PROGRAM ControlePID_Ladder
  VAR
    NIVEL_PV_RAW : UINT := 0;
    AUX_NIVEL_PV : REAL := 0;
    AUX_NIVEL_PV0 : REAL := 0;
    VAZAO_ENTRADA_RAW : UINT := 0;
    VALVULA_SAIDA_RAW : UINT := 3500;
    AUTO_MODE_RAW : UINT := 1;
    VAZAO_SAIDA_RAW : UINT := 0;
    PLANTA_STATUS_RAW : UINT := 0;
    SP_RAW : UINT := 5000;
    KP_RAW : UINT := 200;
    TR_RAW : UINT := 120;
    TD_RAW : UINT := 0;
    MANUAL_OUT_RAW : UINT := 2000;
    PID_XOUT_PCT : REAL := 0.0;
    CONTROLE_ENABLE_RAW : UINT := 1;
    RESET_PLANTA_RAW : UINT := 0;
    FALHA_SENSOR_CMD_RAW : UINT := 0;
    BOMBA_DISPONIVEL_CMD_RAW : UINT := 1;
    RESET_PID_RAW : UINT := 0;
    NIVEL_PV_PCT : REAL := 0.0;
    NIVEL_SP_PCT : REAL := 0.0;
    NIVEL_SP_APLICADO_PCT : REAL := 50.0;
    VAZAO_SAIDA_PCT : REAL := 0.0;
    BOMBA_CMD_PCT : REAL := 0.0;
    SP_MAX_PCT : REAL := 80.0;
    SP_MIN_PCT : REAL := 20.0;
    MV_MIN_PCT : REAL := 0.0;
    MV_MAX_PCT : REAL := 85.0;
    GANHO_FF : REAL := 0.8;
    MV_COMPENSACAO_PCT : REAL := 0.0;
    MV_APOS_MAX_PCT : REAL := 0.0;
    MV_LIMITADA_SUP_PCT : REAL := 0.0;
    BOMBA_CMD_RAW : UINT := 0;
    RESTRICAO_ATIVA : BOOL := FALSE;
    PID_SATURADO : BOOL := FALSE;
    SENSOR_FAULT : BOOL := FALSE;
    PID_ACTIVE : BOOL := FALSE;
    BOMBA_DISPONIVEL_FB : BOOL := TRUE;
    PLANTA_ENABLE_FB : BOOL := TRUE;
    FALHA_SENSOR_FB : BOOL := FALSE;
    PID_KP : REAL := 2.0;
    PID_TR : REAL := 12.0;
    PID_TD : REAL := 0.0;
    AUX_NIVEL_SP : REAL := 0.0;
    AUX_MAX_SP : REAL := 0.0;
    AUX_VAZAO_SAIDA : REAL := 0.0;
    AUX_VAZAO_SAIDA0 : REAL := 0.0;
    AUX : REAL;
    AUX_DIF_RESTRICAO : REAL := 0.0;
    CICLO_PID : TIME := T#100ms;
    AUX_BOMBA_CMD : REAL := 0.0;
    PID0 : PID;
  END_VAR
  VAR  (* added by the conversion: wires and edge detectors of the diagram *)
    _MAX19_OUT : REAL;
  END_VAR

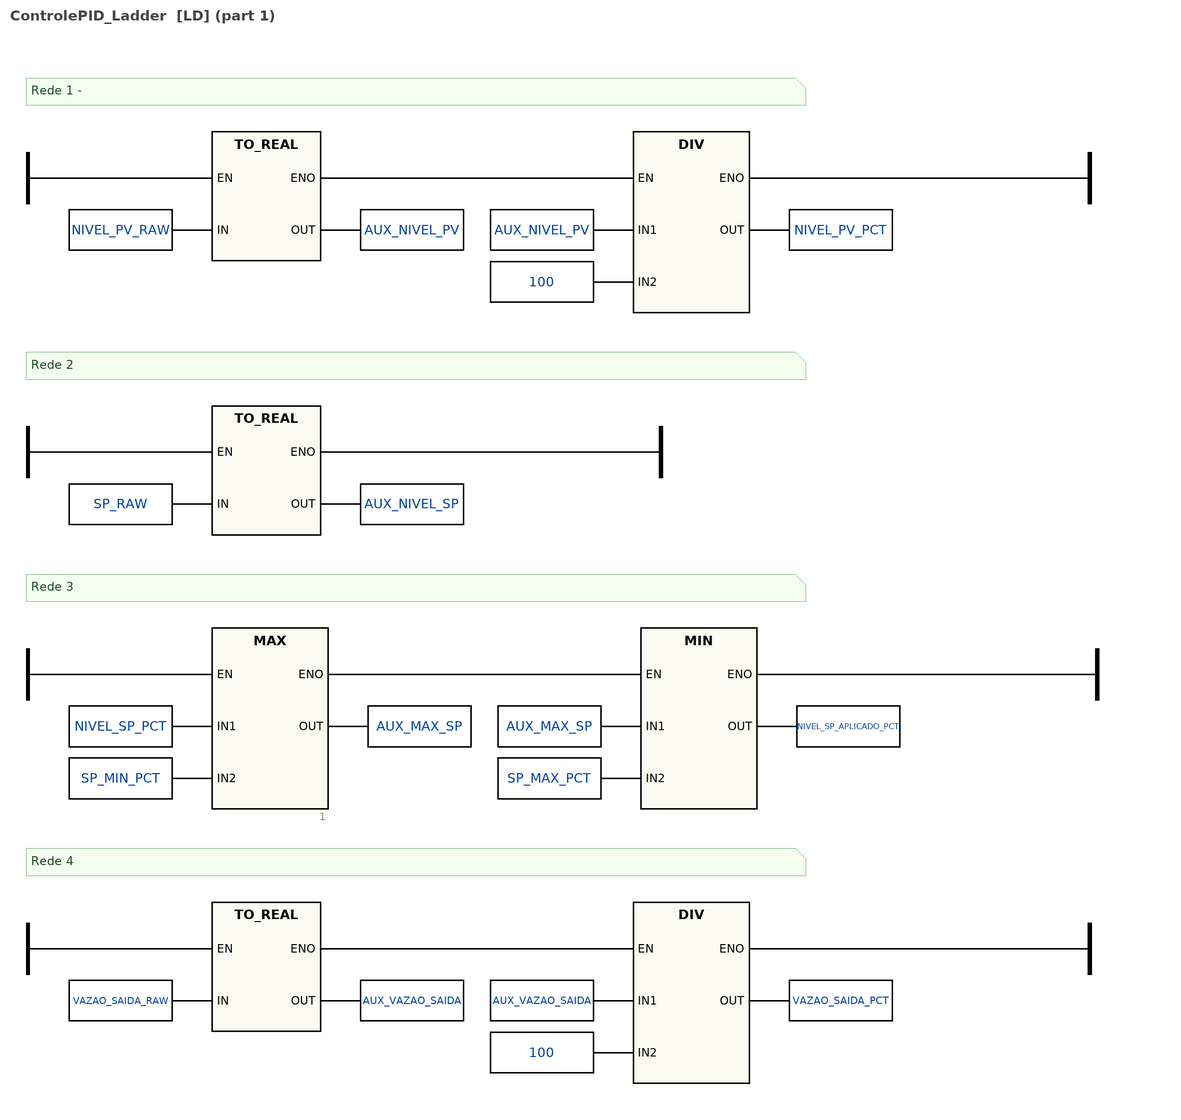
(* LD diagram, written out as Structured Text *)
(* Rede 1 - *)
(* Rede 2 *)
(* Rede 3 *)
_MAX19_OUT := MAX(NIVEL_SP_PCT, SP_MIN_PCT);
AUX_NIVEL_PV := TO_REAL(NIVEL_PV_RAW);
NIVEL_PV_PCT := AUX_NIVEL_PV / 100;
AUX_NIVEL_SP := TO_REAL(SP_RAW);
AUX_MAX_SP := _MAX19_OUT;
NIVEL_SP_APLICADO_PCT := MIN(AUX_MAX_SP, SP_MAX_PCT);
(* Rede 4 *)
AUX_VAZAO_SAIDA := TO_REAL(VAZAO_SAIDA_RAW);
VAZAO_SAIDA_PCT := AUX_VAZAO_SAIDA / 100;
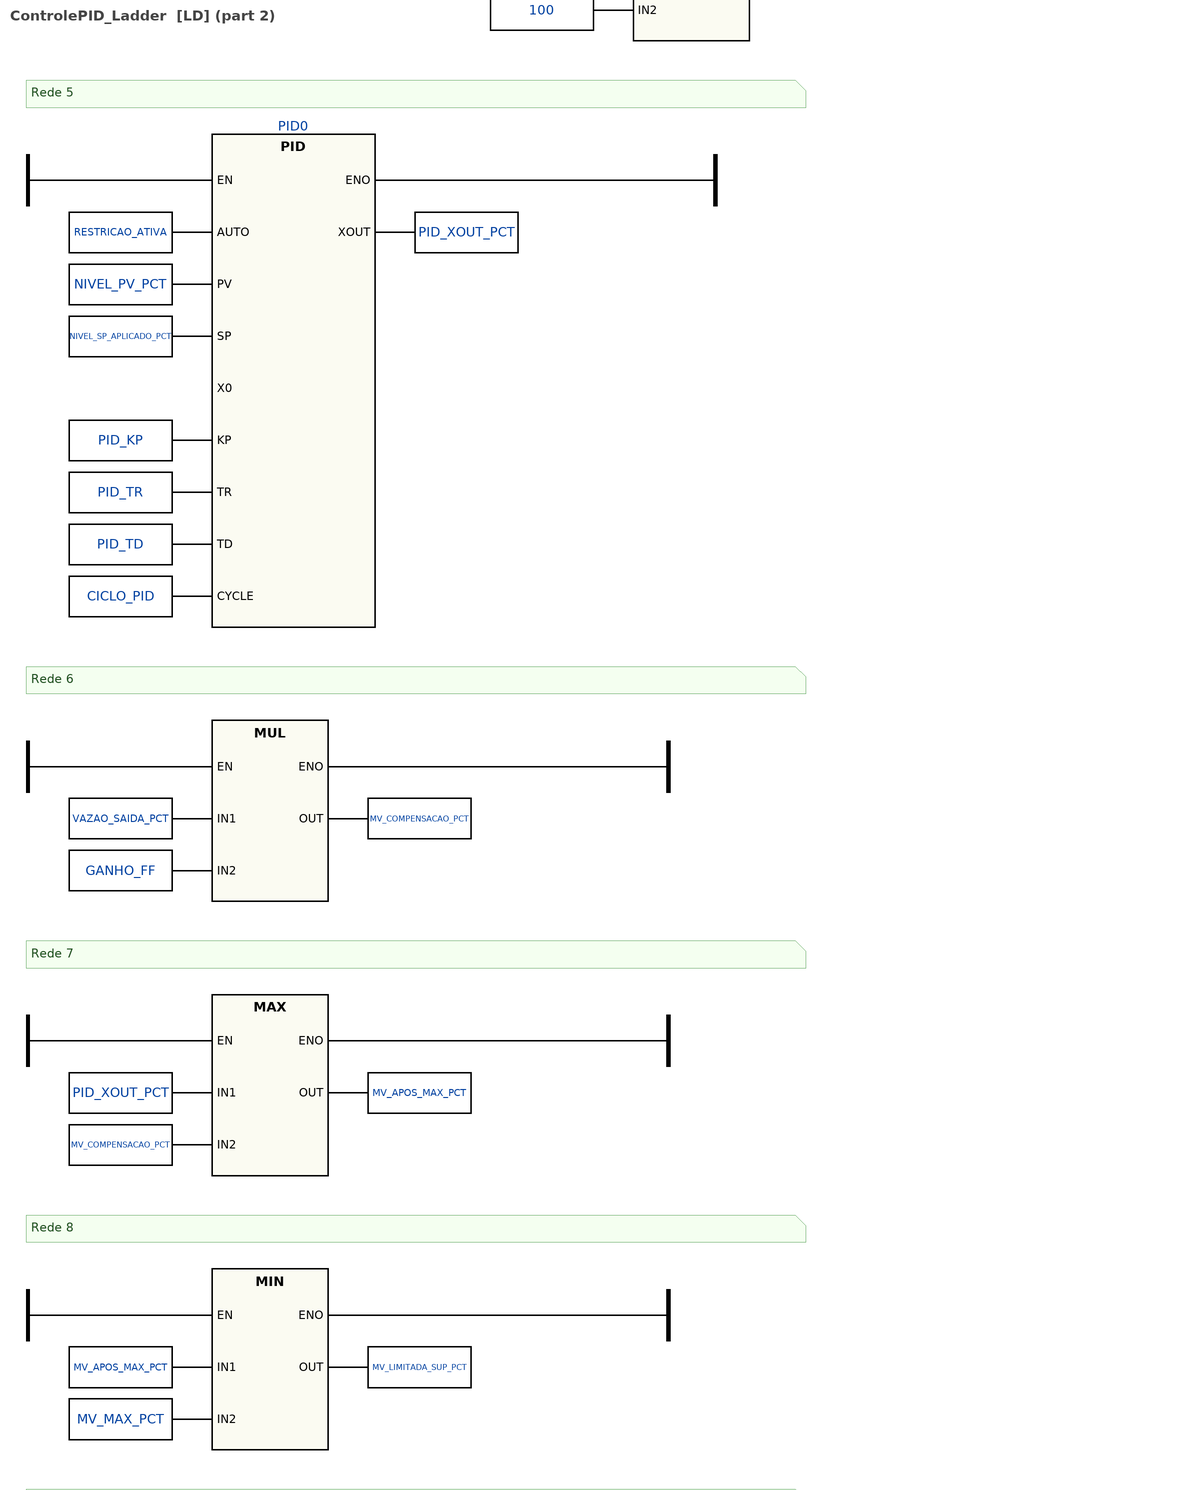
(* Rede 5 *)
PID0(AUTO := RESTRICAO_ATIVA, PV := NIVEL_PV_PCT, SP := NIVEL_SP_APLICADO_PCT, KP := PID_KP, TR := PID_TR, TD := PID_TD, CYCLE := CICLO_PID);
PID_XOUT_PCT := PID0.XOUT;
(* Rede 6 *)
MV_COMPENSACAO_PCT := VAZAO_SAIDA_PCT * GANHO_FF;
(* Rede 7 *)
MV_APOS_MAX_PCT := MAX(PID_XOUT_PCT, MV_COMPENSACAO_PCT);
(* Rede 8 *)
MV_LIMITADA_SUP_PCT := MIN(MV_APOS_MAX_PCT, MV_MAX_PCT);
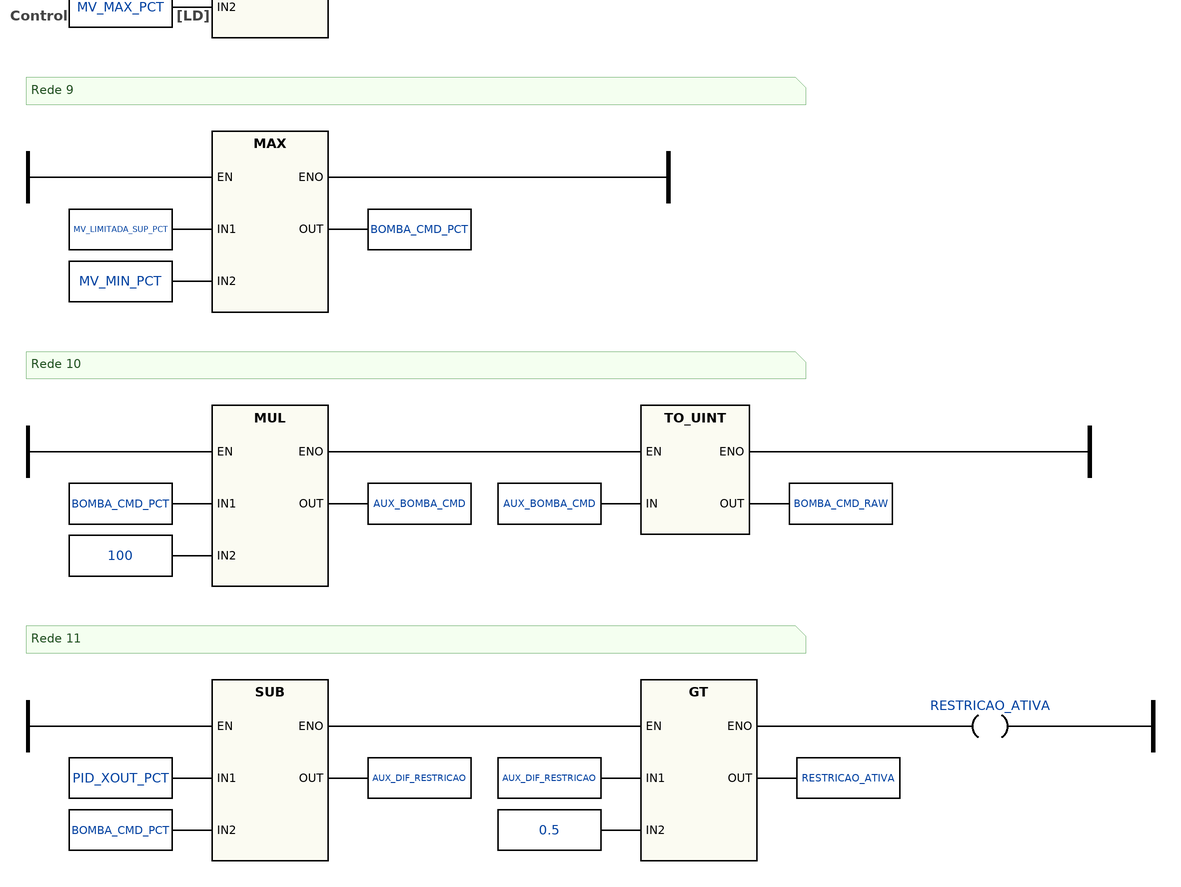
(* Rede 9 *)
BOMBA_CMD_PCT := MAX(MV_LIMITADA_SUP_PCT, MV_MIN_PCT);
(* Rede 10 *)
AUX_BOMBA_CMD := BOMBA_CMD_PCT * 100;
BOMBA_CMD_RAW := TO_UINT(AUX_BOMBA_CMD);
(* Rede 11 *)
RESTRICAO_ATIVA := TRUE;
AUX_DIF_RESTRICAO := PID_XOUT_PCT - BOMBA_CMD_PCT;
RESTRICAO_ATIVA := AUX_DIF_RESTRICAO > 0.5;
END_PROGRAM
